// TIA Portal V19 export
VAR_GLOBAL   // PLC tag table "Default tag table"
   "EMG STOP-1" AT %I0.0 : Bool;
   "EMG STOP-2" AT %I0.1 : Bool;
   "HOOTER RESET-1" AT %I0.2 : Bool;
   "HOOTER RESET-2" AT %I0.3 : Bool;
   "MFG AIR PRESSURE SWITCH" AT %I0.4 : Bool;
   "PHASE FAIL" AT %I0.5 : Bool;
   "MFG VESSEL MOTOR TRIP" AT %I0.6 : Bool;
   "PREMIXING VESSEL MOTOR TRIP" AT %I0.7 : Bool;
   "STORAGE VESSEL-1 MOTOR TRIP" AT %I1.0 : Bool;
   "STORAGE VESSEL-2 MOTOR TRIP" AT %I1.1 : Bool;
   "INLINE HOMOGENIZER-1 TRIP" AT %I1.2 : Bool;
   "FILTER PRESS MOTOR TRIP" AT %I1.3 : Bool;
   "INLINE HOMOGENIZER-2 TRIP" AT %I1.4 : Bool;
   "MFG LOBE PUMP TRIP" AT %I1.5 : Bool;
   "STORAGE VESSEL-1 LOBE PUMP TRIP" AT %I1.6 : Bool;
   "STORAGE VESSEL-2 LOBE PUMP TRIP" AT %I1.7 : Bool;
   "SUGAR VESSEL MOTOR TRIP" AT %I2.0 : Bool;
   "BASKET FILTER MOTOR TRIP" AT %I2.1 : Bool;
   "VACUUME PUMP-1 TRIP" AT %I2.2 : Bool;
   "VACUUME PUMP-2 TRIP" AT %I2.3 : Bool;
   "CIP FORWARD PUMP TRIP" AT %I2.4 : Bool;
   "CIP REVERSE PUMP TRIP" AT %I2.5 : Bool;
   "LEVEL SWITCH LOW-ALKALI" AT %I2.6 : Bool;
   "LEVEL SWITCH HIGH-ALKALI" AT %I2.7 : Bool;
   "LEVEL SWITCH LOW-ACID" AT %I3.0 : Bool;
   "LEVEL SWITCH HIGH-ACID" AT %I3.1 : Bool;
   "FLOW SWITCH- MFG" AT %I3.2 : Bool;
   "FLOW SWITCH- PREMIXING" AT %I3.3 : Bool;
   "FLOW SWITCH- STORAGE VESSEL-1" AT %I3.4 : Bool;
   "FLOW SWITCH- STORAGE VESSEL-2" AT %I3.5 : Bool;
   "FLOW SWITCH- SUGAR VESSEL" AT %I3.6 : Bool;
   "FLOW SWITCH- INLINE HMOGENIZER-1" AT %I3.7 : Bool;
   "FLOW SWITCH- INLINE HMOGENIZER-2" AT %I4.0 : Bool;
   "LEVEL FLOW SWITCH-1" AT %I4.1 : Bool;
   "LEVEL FLOW SWITCH-2" AT %I4.2 : Bool;
   "SUGAR AIR PRESSURE SWITCH" AT %I4.3 : Bool;
   "DI SPARE_1" AT %I4.4 : Bool;
   "DI SPARE_2" AT %I4.5 : Bool;
   "DI SPARE_3" AT %I4.6 : Bool;
   "DI SPARE_4" AT %I4.7 : Bool;
   "HOOTER-1" AT %Q0.0 : Bool;
   "HOOTER-2" AT %Q0.1 : Bool;
   "MFG VESSEL MOTOR" AT %Q0.2 : Bool;
   "PREMIXING VESSEL MOTOR" AT %Q0.3 : Bool;
   "STORAGE VESSEL-1 MOTOR" AT %Q0.4 : Bool;
   "STORAGE VESSEL-2 MOTOR" AT %Q0.5 : Bool;
   "INLINE HOMOGENIZER-1" AT %Q0.6 : Bool;
   "FILTER PRESS MOTOR" AT %Q0.7 : Bool;
   "INLINE HOMOGENIZER-2" AT %Q1.0 : Bool;
   "MFG LOBE PUMP" AT %Q1.1 : Bool;
   "STORAGE VESSEL-1 LOBE PUMP" AT %Q1.2 : Bool;
   "STORAGE VESSEL-2 LOBE PUMP" AT %Q1.3 : Bool;
   "SUGAR VESSEL MOTOR" AT %Q1.4 : Bool;
   "BASKET FILTER MOTOR" AT %Q1.5 : Bool;
   "VACUUME PUMP-1" AT %Q1.6 : Bool;
   "VACUUME PUMP-2" AT %Q1.7 : Bool;
   "CIP FORWARD PUMP" AT %Q2.0 : Bool;
   "CIP REVERSE PUMP" AT %Q2.1 : Bool;
   "DOSING PUMP-1 ALKALI" AT %Q2.2 : Bool;
   "DOSING PUMP-2 ACID" AT %Q2.3 : Bool;
   "MFG VESSEL LAMP" AT %Q2.4 : Bool;
   "PREMIXING VESSEL LAMP" AT %Q2.5 : Bool;
   "STORAGE VESSEL-1 LAMP" AT %Q2.6 : Bool;
   "STORAGE VESSEL-2 LAMP" AT %Q2.7 : Bool;
   "SUGAR VESSEL LAMP" AT %Q3.0 : Bool;
   "PBV-01 ON SUGAR SUCTION LINE" AT %Q3.1 : Bool;
   "PBV- 02 ON VACUUM INLET LINE" AT %Q3.2 : Bool;
   "PBV- 03 ON VENT FILTER" AT %Q3.3 : Bool;
   "PAV- 03 ON AIR INLET LINE" AT %Q3.4 : Bool;
   "PBV- 04 FROM BOTTOM OUTLET TO CIP INLET LINE" AT %Q3.5 : Bool;
   "PBV- 05 ON SPRAY BALL INLET LINE" AT %Q3.6 : Bool;
   "PBV- 06 ON PW INLET LINE" AT %Q3.7 : Bool;
   "PBV- 07 ON VACUUM VENT LINE" AT %Q4.0 : Bool;
   "PAV- 07 ON SEAL COOLING INLET LINE FOR STIRRER" AT %Q4.1 : Bool;
   "PAV- 08 ON AIR INLET LINE" AT %Q4.2 : Bool;
   "PAV- 09 ON STEAM INLET LINE" AT %Q4.3 : Bool;
   "PAV- 10 ON STEAM OUTLET LINE" AT %Q4.4 : Bool;
   "PAV- 11 ON SEAL COOLING INLET LINE" AT %Q4.5 : Bool;
   "PBV- 12 FROM BOTTOM OUTLET TO CIP DRAIN LINE" AT %Q4.6 : Bool;
   "PBV- 13 FROM BOTTOM OUTLET TO CIP INLET LINE" AT %Q4.7 : Bool;
   "PBV- 14 ON BOTTOM OUTLET LINE" AT %Q5.0 : Bool;
   "PBV- 15 FROM BOTTOM OUTLET TO DRAIN LINE" AT %Q5.1 : Bool;
   "PBV- 16 FROM BOTTOM OUTLET TO BASKET FILTER INLET LINE" AT %Q5.2 : Bool;
   "PBV- 17 ON BASKET FILTER INLET LINE" AT %Q5.3 : Bool;
   "PBV- 18 ON BASKET FILTER OUTLET LINE" AT %Q5.4 : Bool;
   "PBV- 19 ON SUGAR VESSEL CIP INLET LINE" AT %Q5.5 : Bool;
   "PBV- 20 ON PREMIXING VESEL CIP INLET LINE" AT %Q5.6 : Bool;
   "PBV- 21 ON PW INLET BYPASS LINE" AT %Q5.7 : Bool;
   "PBV- 22 ON PW INLET LINE" AT %Q6.0 : Bool;
   "PBV- 23 ON VENT FILTER" AT %Q6.1 : Bool;
   "PBV- 24 ON VACUUM INLET LINE" AT %Q6.2 : Bool;
   "PBV- 25 FROM BOTTOM OUTLET TO SPRAY BALL INLET LINE" AT %Q6.3 : Bool;
   "PBV- 26 ON SPRAY BALL INLET LINE" AT %Q6.4 : Bool;
   "PBV- 27 FROM SUGAR TO PREMIXING VESSEL INLET LINE" AT %Q6.5 : Bool;
   "PBV- 28 ON VESSEL TOP DISH" AT %Q6.6 : Bool;
   "PBV- 29 ON RECIRCULATION LINE" AT %Q6.7 : Bool;
   "PBV- 30 FROM PREMIXING TO STORAGE TRANSFER LINE" AT %Q7.0 : Bool;
   "PBV- 31 FROM SORBITOL VESSEL TO PREMIXING VESSEL TRANSFER LINE" AT %Q7.1 : Bool;
   "PBV- 32 FROM PREMIXING TO MFG TRANSFER LINE" AT %Q7.2 : Bool;
   "PAV- 33 ON STEAM INLET LINE" AT %Q7.3 : Bool;
   "PAV- 35 ON COOLING WATER OUTLET LINE" AT %Q7.4 : Bool;
   "PAV- 36 ON STEAM OUTLET LINE" AT %Q7.5 : Bool;
   "PAV- 37 ON BYPASS CONDENSATE LINE" AT %Q7.6 : Bool;
   "PAV- 38 ON COOLING WATER INLET LINE" AT %Q7.7 : Bool;
   "PBV- 39 FROM BOTTOM OUTLET TO SPRAY BALL INLET LINE" AT %Q8.0 : Bool;
   "PBV- 40 FROM BOTTOM OUTLET TO SPRAY BALL INLET LINE" AT %Q8.1 : Bool;
   "PBV- 41 FROM BOTTOM OUTLET TO DRAIN LINE" AT %Q8.2 : Bool;
   "PBV- 42 FROM BOTTOM OUTLET TO DRAIN LINE" AT %Q8.3 : Bool;
   "PBV- 43 FROM BOTTOM OUTLET TO INLINE HOMOGENIZER LINE" AT %Q8.4 : Bool;
   "PBV- 44 FROM VESSEL OUTLET TO FILTER PRESS LINE" AT %Q8.5 : Bool;
   "PBV- 45 FROM INLINE HOMOGENIZER TO STORAGE TRANSFER LINE" AT %Q8.6 : Bool;
   "PBV- 46 ON INLINE HOMOGENIZER INLET LINE" AT %Q8.7 : Bool;
   "PBV- 47 ON INLINE HOMOGENIZER RECIRCULATION LINE" AT %Q9.0 : Bool;
   "PAV- 48 ON SEAL COOLING INLET LINE FOR INLINE HOMOGENIZER" AT %Q9.1 : Bool;
   "PBV- 49 INLINE HOMOGENIZER DRAIN LINE" AT %Q9.2 : Bool;
   "PBV- 50 ON PW INLET LINE" AT %Q9.3 : Bool;
   "PBV- 51 FROM PW INLET TO DRAIN LINE" AT %Q9.4 : Bool;
   "PBV- 52 FROM SUGAR MELTING TO MFG VESSEL TRANSFER LINE" AT %Q9.5 : Bool;
   "PBV- 53 ON VENT FILTER" AT %Q9.6 : Bool;
   "PBV- 54 FROM BOTTOM OUTLET TO SPRAY BALL INLET LINE" AT %Q9.7 : Bool;
   "PBV- 55 ON SPRAY BALL INLET LINE" AT %Q10.0 : Bool;
   "PBV- 56 ON VACUUM INLET LINE" AT %Q10.1 : Bool;
   "PBV- 57 ON RECIRCULATION LINE" AT %Q10.2 : Bool;
   "PBV- 58 FROM INLINE HOMOGENIZER TO STORAGE TRANSFER LINE" AT %Q10.3 : Bool;
   "PBV- 59 FROM PREMIXING TO FILTER PRESS TRANSFER LINE" AT %Q10.4 : Bool;
   "PBV- 60 FROM PREMIXING LOBE PUMP TO FILTER PRESS LINE" AT %Q10.5 : Bool;
   "PAV- 61 ON COOLING OUTLET LINE" AT %Q10.6 : Bool;
   "PAV- 62 ON STEAM INLET LINE" AT %Q10.7 : Bool;
   "PAV- 63 ON COOLING INLET LINE" AT %Q11.0 : Bool;
   "PAV- 64 ON SEAL COOLING INLET LINE FOR STIRRER" AT %Q11.1 : Bool;
   "PAV- 65 ON STEAM OUTLET LINE" AT %Q11.2 : Bool;
   "PAV- 66 ON BYPASS CONDENSATE LINE" AT %Q11.3 : Bool;
   "PBV- 67 FROM BOTTOM OUTLET TO SPRAY BALL INLET LINE" AT %Q11.4 : Bool;
   "PBV- 68 FROM BOTTOM OUTLET TO SPRAY BALL INLET LINE" AT %Q11.5 : Bool;
   "PBV- 69 FROM BOTTOM OUTLET TO DRAIN LINE" AT %Q11.6 : Bool;
   "PBV- 70 FROM BOTTOM OUTLET TO DRAIN LINE" AT %Q11.7 : Bool;
   "PBV- 71 FROM BOTTOM OUTLET TO INLINE HOMOGENIZER LINE" AT %Q12.0 : Bool;
   "PBV- 72 ON INLINE HOMOGENIZER INLET LINE" AT %Q12.1 : Bool;
   "PBV- 73 ON RECIRCULATION LINE" AT %Q12.2 : Bool;
   "PBV- 74 FROM BOTTOM OUTLET TO INLINE HOMOGENIZER LINE" AT %Q12.3 : Bool;
   "PAV- 75 ON SEAL COOLING INLET LINE FOR HOMOGENIZER" AT %Q12.4 : Bool;
   "PBV- 76 FROM INLINE HOMOGENIZER TO DRAIN LINE" AT %Q12.5 : Bool;
   "PBV- 77 ON FILTER PRESS INLET LINE" AT %Q12.6 : Bool;
   "PBV- 78 ON FILTER PRESS OUTLET LINE" AT %Q12.7 : Bool;
   "PBV- 79 ON FILTER PRESS OUTLET LINE" AT %Q13.0 : Bool;
   "PBV- 80 FROM MFG TO STORAGE VESSEL TRANSFER LINE" AT %Q13.1 : Bool;
   "PBV- 81 ON VESSEL TOP DISH" AT %Q13.2 : Bool;
   "PBV- 82 FROM BOTTOM OUTLET TO SPRAY BALL INLET LINE" AT %Q13.3 : Bool;
   "PBV- 83 ON CIP INLET LINE" AT %Q13.4 : Bool;
   "PAV- 84 ON SEAL COOLING LINE OF BOTTOM STIRRER" AT %Q13.5 : Bool;
   "PBV- 85 FROM BOTTOM OUTLET TO SPRAY BALL INLET LINE" AT %Q13.6 : Bool;
   "PBV- 86 FROM BOTTOM OUTLET TO DRAIN LINE" AT %Q13.7 : Bool;
   "PBV- 87 FROM BOTTOM OUTLET TO SPRAY BALL INLET LINE" AT %Q14.0 : Bool;
   "PBV- 88 FROM BOTTOM OUTLET TO DRAIN LINE" AT %Q14.1 : Bool;
   "PBV- 89 FROM VESSEL BOTTOM OUTLET TO LOBE PUMP LINE" AT %Q14.2 : Bool;
   "PBV- 90 ON VESSEL TOP DISH" AT %Q14.3 : Bool;
   "PBV- 91 FROM BOTTOM OUTLET TO SPRAY BALL INLET LINE" AT %Q14.4 : Bool;
   "PBV- 92 ON SPRAY BALL INLET LINE" AT %Q14.5 : Bool;
   "PAV- 93 ON SEAL COOLING LINE OF BOTTOM STIRRER" AT %Q14.6 : Bool;
   "PBV- 94 FROM BOTTOM OUTLET TO SPRAY BALL INLET LINE" AT %Q14.7 : Bool;
   "PBV- 95 FROM BOTTOM OUTLET TO DRAIN LINE" AT %Q15.0 : Bool;
   "PBV- 96 FROM BOTTOM OUTLET TO SPRAY BALL INLET LINE" AT %Q15.1 : Bool;
   "PBV- 97 FROM BOTTOM OUTLET TO DRAIN LINE" AT %Q15.2 : Bool;
   "PBV- 98 FROM BOTTOM OUTLET TO LOBE PUMP LINE" AT %Q15.3 : Bool;
   "PBV- 99 ON VACUUM VENT LINE" AT %Q15.4 : Bool;
   "PFBV- 100 ON VESSEL BOTTOM DISH" AT %Q15.5 : Bool;
   "PFBV- 101 ON VESSEL BOTTOM DISH" AT %Q15.6 : Bool;
   "PFBV- 102 ON VESSEL BOTTOM DISH" AT %Q15.7 : Bool;
   "PFBV- 103 ON VESSEL BOTTOM DISH" AT %Q16.0 : Bool;
   "PFBV- 104 ON VESSEL BOTTOM DISH" AT %Q16.1 : Bool;
   "PAV- 105 ON AIR INLET LINE" AT %Q16.2 : Bool;
   "DO SPARE_1" AT %Q16.3 : Bool;
   "DO SPARE_2" AT %Q16.4 : Bool;
   "DO SPARE_3" AT %Q16.5 : Bool;
   "DO SPARE_4" AT %Q16.6 : Bool;
   "DO SPARE_5" AT %Q16.7 : Bool;
   "DO SPARE_6" AT %Q17.0 : Bool;
   "DO SPARE_7" AT %Q17.1 : Bool;
   "DO SPARE_8" AT %Q17.2 : Bool;
   "DO SPARE_9" AT %Q17.3 : Bool;
   "DO SPARE_10" AT %Q17.4 : Bool;
   "DO SPARE_11" AT %Q17.5 : Bool;
   "DO SPARE_12" AT %Q17.6 : Bool;
   "DO SPARE_13" AT %Q17.7 : Bool;
   "DO SPARE_14" AT %Q18.0 : Bool;
   "DO SPARE_15" AT %Q18.1 : Bool;
   "DO SPARE_16" AT %Q18.2 : Bool;
   "DO SPARE_17" AT %Q18.3 : Bool;
   "DO SPARE_18" AT %Q18.4 : Bool;
   "DO SPARE_19" AT %Q18.5 : Bool;
   "DO SPARE_20" AT %Q18.6 : Bool;
   "DO SPARE_21" AT %Q18.7 : Bool;
   "DO SPARE_22" AT %Q19.0 : Bool;
   "DO SPARE_23" AT %Q19.1 : Bool;
   "DO SPARE_24" AT %Q19.2 : Bool;
   "DO SPARE_25" AT %Q19.3 : Bool;
   "DO SPARE_26" AT %Q19.4 : Bool;
   "DO SPARE_27" AT %Q19.5 : Bool;
   "DO SPARE_28" AT %Q19.6 : Bool;
   "DO SPARE_29" AT %Q19.7 : Bool;
   "DO SPARE_30" AT %Q20.0 : Bool;
   "DO SPARE_31" AT %Q20.1 : Bool;
   "DO SPARE_32" AT %Q20.2 : Bool;
   "DO SPARE_33" AT %Q20.3 : Bool;
   "DO SPARE_34" AT %Q20.4 : Bool;
   "DO SPARE_35" AT %Q20.5 : Bool;
   "DO SPARE_36" AT %Q20.6 : Bool;
   "DO SPARE_37" AT %Q20.7 : Bool;
   "DO SPARE_38" AT %Q21.0 : Bool;
   "DO SPARE_39" AT %Q21.1 : Bool;
   "DO SPARE_40" AT %Q21.2 : Bool;
   "DO SPARE_41" AT %Q21.3 : Bool;
   "DO SPARE_42" AT %Q21.4 : Bool;
   "DO SPARE_43" AT %Q21.5 : Bool;
   "DO SPARE_44" AT %Q21.6 : Bool;
   "DO SPARE_45" AT %Q21.7 : Bool;
   "LOAD CELL- MFG" AT %IW5 : Int;
   "LOAD CELL- PREMIXING" AT %IW7 : Int;
   "LOAD CELL- SUGAR" AT %IW9 : Int;
   "LOAD CELL- STORAGE-1" AT %IW11 : Int;
   "LOAD CELL- STORAGE-2" AT %IW13 : Int;
   "CONDUCTIVITY METER" AT %IW15 : Int;
   "TEMP.SENSOR- MFG INLET" AT %IW17 : Int;
   "TEMP.SENSOR- MFG PRODUCT" AT %IW19 : Int;
   "TEMP.SENSOR- PREMIXING INLET" AT %IW21 : Int;
   "TEMP.SENSOR- PREMIXING PRODUCT" AT %IW23 : Int;
   "TEMP.SENSOR- SUGAR INLET" AT %IW25 : Int;
   "TEMP.SENSOR- SUGAR PRODUCT" AT %IW27 : Int;
   "TEMP.SENSOR- CIP1" AT %IW29 : Int;
   "PRESSURE TRANSMTER- MFG AIRINLET" AT %IW31 : Int;
   "PRESSURE TRANSMTER- SUGAR AIRINLET" AT %IW33 : Int;
   "VACUUME TRANSMTER- MFG" AT %IW35 : Int;
   "VACUUME TRANSMTER- SUGAR" AT %IW37 : Int;
   "VACUUME TRANSMTER- PREMIXING" AT %IW39 : Int;
   "TEMP.SENSOR CIP2" AT %IW41 : Int;
   "AI SPARE_1" AT %IW43 : Int;
   "AI SPARE_2" AT %IW45 : Int;
   "AI SPARE_3" AT %IW47 : Int;
   "AI SPARE_4" AT %IW49 : Int;
   "AI SPARE_5" AT %IW51 : Int;
   "MFG VESSEL MOTOR SPEED" AT %QW22 : Int;
   "PREMIXING VESSEL MOTOR SPEED" AT %QW24 : Int;
   "STORAGE VESSEL-1 MOTOR SPEED" AT %QW26 : Int;
   "STORAGE VESSEL-2 MOTOR SPEED" AT %QW28 : Int;
   "SUGAR VESSEL MOTOR SPEED" AT %QW30 : Int;
   "AO SPARE_1" AT %QW32 : Int;
   "AO SPARE_2" AT %QW34 : Int;
   "AO SPARE_3" AT %QW36 : Int;
   Tag_1 AT %IW3 : Word;
   System_Byte AT %MB1 : Byte;
   FirstScan AT %M1.0 : Bool;
   DiagStatusUpdate AT %M1.1 : Bool;
   AlwaysTRUE AT %M1.2 : Bool;
   AlwaysFALSE AT %M1.3 : Bool;
   Clock_Byte AT %MB0 : Byte;
   Clock_10Hz AT %M0.0 : Bool;
   Clock_5Hz AT %M0.1 : Bool;
   "Clock_2.5Hz" AT %M0.2 : Bool;
   Clock_2Hz AT %M0.3 : Bool;
   "Clock_1.25Hz" AT %M0.4 : Bool;
   Clock_1Hz AT %M0.5 : Bool;
   "Clock_0.625Hz" AT %M0.6 : Bool;
   "Clock_0.5Hz" AT %M0.7 : Bool;
END_VAR
